Yaskawa INFORM job: B-6-08279-80-0-R.JBI

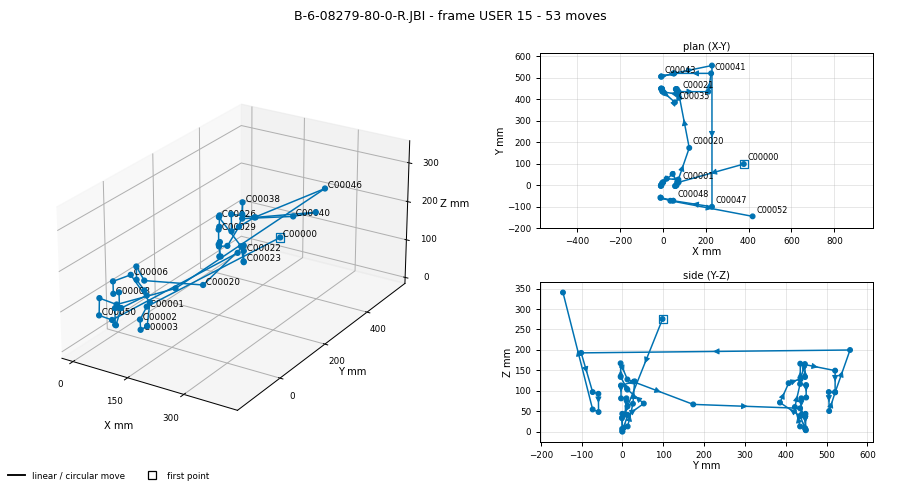
[picture p0: tool path of B-6-08279-80-0-R.JBI in frame USER 15, 53 of 53 moves have a stored position in this frame; points joined in program order, loops and branches not executed]
/JOB
//NAME B-6-08279-80-0-R
///FOLDERNAME PART_420-08279-80
//POS
///NPOS 53,0,53,0,0,0
///USER 15
///TOOL 4
///POSTYPE USER
///RECTAN
///RCONF 1,0,0,0,0,0,0,0,0,0,0,0,0,0,0,0,0,0,0,0,0,0,0,0
C00000=377.977,98.282,275.548,-96.7918,26.0599,130.3916
C00001=73.206,12.887,62.532,-108.1130,33.6440,124.7280
C00002=63.428,-1.162,32.750,-108.1127,33.6388,124.7316
C00003=64.140,-0.660,6.535,-108.1124,33.6386,124.7313
C00004=73.207,12.886,12.496,-108.1130,33.6440,124.7280
C00005=73.209,25.753,68.034,-108.1130,33.6440,124.7280
C00006=18.285,29.861,123.023,-105.1660,8.3780,132.7380
C00007=-8.546,-3.528,112.950,-105.6931,27.7436,134.0533
C00008=-8.576,-3.348,81.228,-105.6913,27.7455,134.0523
C00009=-1.744,9.833,81.413,-106.8820,26.9670,127.1640
C00010=-1.744,9.833,41.151,-106.8820,26.9670,127.1640
C00011=-7.181,-0.325,43.460,-123.9089,34.0116,115.6065
C00012=-7.814,-0.185,0.775,-124.5345,34.0910,114.8301
C00013=-5.856,-0.182,-0.179,-124.5337,34.0915,114.8299
C00014=1.309,12.886,40.637,-115.9500,15.0640,123.8880
C00015=46.568,52.366,68.637,-115.9500,15.0640,123.8880
C00016=68.126,12.203,102.713,-51.9240,65.1860,170.4170
C00017=58.125,-4.227,133.697,-54.9585,64.7745,167.3122
C00018=58.441,-4.415,167.108,-54.9570,64.7753,167.3130
C00019=68.127,12.203,127.579,-51.9240,65.1860,170.4170
C00020=123.702,173.377,66.504,-51.9240,65.1860,170.4170
C00021=73.207,435.046,56.988,108.1130,33.6440,-124.7280
C00022=65.557,447.328,36.164,107.9786,34.0375,-124.0036
C00023=65.003,447.488,7.952,107.9788,34.0378,-124.0032
C00024=73.207,435.046,12.497,108.1130,33.6440,-124.7280
C00025=73.208,422.239,60.087,108.1130,33.6440,-124.7280
C00026=1.310,435.046,116.590,106.4700,24.0930,-128.1180
C00027=-6.306,449.805,113.929,105.8852,24.7458,-131.5857
C00028=-7.382,449.972,83.303,105.8852,24.7463,-131.5846
C00029=-1.744,438.100,81.414,106.4700,24.0930,-128.1180
C00030=-1.744,438.100,41.152,106.4700,24.0930,-128.1180
C00031=-4.715,448.204,43.414,105.1850,25.4207,-135.4134
C00032=-6.772,448.950,3.270,120.3972,28.6468,-129.7143
C00033=-2.895,448.940,4.238,120.3976,28.6469,-129.7144
C00034=1.310,435.046,37.856,114.8060,13.4990,-125.4170
C00035=56.824,385.802,71.014,114.8060,13.4990,-125.4170
C00036=76.829,406.941,118.422,51.9240,65.1860,-170.4170
C00037=61.206,447.085,133.435,51.9129,65.1891,-170.4230
C00038=62.176,446.887,165.295,51.9216,65.1869,-170.4154
C00039=68.127,435.729,127.579,51.9240,65.1860,-170.4170
C00040=212.373,435.445,166.233,51.9240,65.1860,-170.4170
C00041=225.757,520.809,149.229,-64.9600,52.3020,155.2860
C00042=54.000,520.810,96.661,-64.9600,52.3020,155.2860
C00043=-7.076,505.350,96.754,-64.9604,52.3028,155.2850
C00044=-7.131,506.216,50.245,-64.9620,52.3017,155.2850
C00045=50.732,520.809,95.877,-64.9600,52.3020,155.2860
C00046=229.531,557.327,199.687,42.3120,70.9810,-117.7980
C00047=229.653,-100.956,192.660,69.2460,43.0800,-149.5110
C00048=49.647,-72.877,96.659,69.2460,43.0800,-149.5110
C00049=-8.287,-58.810,92.522,69.2472,43.0782,-149.5115
C00050=-10.780,-58.382,47.854,69.2478,43.0783,-149.5120
C00051=35.736,-72.877,54.138,69.2460,43.0800,-149.5110
C00052=418.971,-145.560,340.461,69.2481,43.0799,-149.5077
///TOOL 0
///POSTYPE ANGLE
///ANGLE
EC00000=15.0000
///TOOL 4
EC00001=15.0000
///TOOL 0
EC00002=15.0000
EC00003=15.0000
///TOOL 4
EC00004=15.0000
EC00005=15.0000
EC00006=15.0000
///TOOL 0
EC00007=15.0000
EC00008=15.0000
///TOOL 4
EC00009=15.0000
EC00010=15.0000
///TOOL 0
EC00011=15.0000
EC00012=15.0000
EC00013=15.0000
///TOOL 4
EC00014=15.0000
EC00015=15.0000
EC00016=15.0000
///TOOL 0
EC00017=15.0000
EC00018=15.0000
///TOOL 4
EC00019=15.0000
EC00020=15.0000
EC00021=15.0000
///TOOL 0
EC00022=15.0000
EC00023=15.0000
///TOOL 4
EC00024=15.0000
EC00025=15.0000
EC00026=15.0000
///TOOL 0
EC00027=15.0000
EC00028=15.0000
///TOOL 4
EC00029=15.0000
EC00030=15.0000
///TOOL 0
EC00031=15.0000
EC00032=15.0000
EC00033=15.0000
///TOOL 4
EC00034=15.0000
EC00035=15.0000
EC00036=15.0000
///TOOL 0
EC00037=15.0000
EC00038=15.0000
///TOOL 4
EC00039=15.0000
EC00040=15.0000
EC00041=15.0000
EC00042=15.0000
///TOOL 0
EC00043=15.0000
EC00044=15.0000
///TOOL 4
EC00045=15.0000
EC00046=15.0000
EC00047=15.0000
EC00048=15.0000
///TOOL 0
EC00049=15.0000
EC00050=15.0000
///TOOL 4
EC00051=15.0000
///TOOL 0
EC00052=15.0000
//INST
///DATE 2021/10/29 11:36
///ATTR SC,RW,RJ
////FRAME USER 15
///GROUP1 RB1
///GROUP2 ST3
NOP
'Path Start: PP56
MOVJ C00000 VJ=100.00  +MOVJ EC00000
SMOVL C00001 V=1250.0  +MOVJ EC00001
SMOVL C00002 V=300.0  +MOVJ EC00002
ARCON ASF#(953)
SMOVL C00003 V=8.5  +MOVJ EC00003
ARCOF AEF#(953)
SMOVL C00004 V=1250.0  +MOVJ EC00004
SMOVL C00005 V=1250.0  +MOVJ EC00005
'Path End
'Path Start: PP54
SMOVL C00006 V=1250.0  +MOVJ EC00006
SMOVL C00007 V=300.0  +MOVJ EC00007
ARCON ASF#(952)
SMOVL C00008 V=6.3  +MOVJ EC00008
ARCOF AEF#(954)
SMOVL C00009 V=300.0  +MOVJ EC00009
SMOVL C00010 V=300.0  +MOVJ EC00010
SMOVL C00011 V=300.0  +MOVJ EC00011
ARCON ASF#(952)
SMOVL C00012 V=6.3  +MOVJ EC00012
SMOVL C00013 V=6.3  +MOVJ EC00013
ARCOF AEF#(954)
SMOVL C00014 V=1250.0  +MOVJ EC00014
SMOVL C00015 V=1250.0  +MOVJ EC00015
'Path End
'Path Start: Path_5
SMOVL C00016 V=1250.0  +MOVJ EC00016
SMOVL C00017 V=1250.0  +MOVJ EC00017
ARCON ASF#(951)
SMOVL C00018 V=8.5  +MOVJ EC00018
ARCOF AEF#(951)
SMOVL C00019 V=1250.0  +MOVJ EC00019
SMOVL C00020 V=1250.0  +MOVJ EC00020
'Path End
'Path Start: PP55
SMOVL C00021 V=1250.0  +MOVJ EC00021
SMOVL C00022 V=300.0  +MOVJ EC00022
ARCON ASF#(952)
SMOVL C00023 V=8.5  +MOVJ EC00023
ARCOF AEF#(952)
SMOVL C00024 V=1250.0  +MOVJ EC00024
SMOVL C00025 V=1250.0  +MOVJ EC00025
'Path End
'Path Start: PP58
SMOVL C00026 V=1250.0  +MOVJ EC00026
SMOVL C00027 V=300.0  +MOVJ EC00027
ARCON ASF#(952)
SMOVL C00028 V=6.3  +MOVJ EC00028
ARCOF AEF#(954)
SMOVL C00029 V=300.0  +MOVJ EC00029
SMOVL C00030 V=300.0  +MOVJ EC00030
SMOVL C00031 V=300.0  +MOVJ EC00031
ARCON ASF#(952)
SMOVL C00032 V=6.3  +MOVJ EC00032
SMOVL C00033 V=6.3  +MOVJ EC00033
ARCOF AEF#(954)
SMOVL C00034 V=1250.0  +MOVJ EC00034
SMOVL C00035 V=1250.0  +MOVJ EC00035
'Path End
'Path Start: Path_4
SMOVL C00036 V=1250.0  +MOVJ EC00036
SMOVL C00037 V=1250.0  +MOVJ EC00037
ARCON ASF#(951)
SMOVL C00038 V=8.5  +MOVJ EC00038
ARCOF AEF#(951)
SMOVL C00039 V=1250.0  +MOVJ EC00039
SMOVL C00040 V=1250.0  +MOVJ EC00040
'Path End
'Path Start: PP57
SMOVL C00041 V=1250.0  +MOVJ EC00041
SMOVL C00042 V=1250.0  +MOVJ EC00042
SMOVL C00043 V=300.0  +MOVJ EC00043
ARCON ASF#(953)
SMOVL C00044 V=8.5  +MOVJ EC00044
ARCOF AEF#(953)
SMOVL C00045 V=1250.0  +MOVJ EC00045
SMOVL C00046 V=1250.0  +MOVJ EC00046
'Path End
'Path Start: PP53
SMOVL C00047 V=1250.0  +MOVJ EC00047
SMOVL C00048 V=1250.0  +MOVJ EC00048
SMOVL C00049 V=300.0  +MOVJ EC00049
ARCON ASF#(953)
SMOVL C00050 V=8.5  +MOVJ EC00050
ARCOF AEF#(953)
SMOVL C00051 V=1250.0  +MOVJ EC00051
SMOVL C00052 V=1250.0  +MOVJ EC00052
'Path End
END
